PROGRAM MAIN
VAR
END_VAR

P_Inputs();
P_Outputs();
P_MachineControl();

END_PROGRAM

(* stored: Version 1.1.0.1, ProductVersion 3.1.4024.11
   POU MAIN: Id {51da1b52-2b53-44ea-a693-73c155047262}, SpecialFunc None *)
